// SIMATIC S7-200 SMART project (STEP 7-Micro/WIN SMART), CPU SR30

SYMBOL_TABLE 表格 1
真空值              VD200
温度值              VD204
罗茨启动真空设定         VD208
罗茨停机真空设定         VD212
温度报警设定           VD216
温度急停设定           VD220
目标真空             VD224
螺杆电流值            VD228
开启清洗电流设定         VD232
关闭清洗电流设定         VD236
频率读取             VW100
电流读取             VW102
频率显示             VW104
电流显示             VW106
频率写入             VW108
手动频率             VW110
清洗时间设定           VW112
吹扫时间设定           VW114
清洗时间显示           VW116
吹扫时间显示           VW118
清洗时间中间量          VW120
吹扫时间中间量          VW122
自动步骤             VW20
延时定时器            T50
流量开关定时器          T51
清洗定时器            T37
吹扫定时器            T38
故障急停             V300.0
故障报警             V300.1
流量开关fault        V300.2
液位开关fault        V300.3
变频器fault         V300.4
罗茨风机过载fault      V300.5
螺杆过载fault        V300.6
急停fault          V300.7
高温报警fault        V301.0
高温急停fault        V301.1
螺杆泵HMI           V500.0
罗茨泵HMI           V500.1
入口阀HMI           V500.2
清洗阀HMI           V500.3
吹扫阀HMI           V500.4
屏蔽蜂鸣器            V500.5
在线清洗HMI          V500.6
END_SYMBOL_TABLE

SYMBOL_TABLE 系统符号
Always_On        SM0.0    // 始终接通
First_Scan_On    SM0.1    // 仅在第一个扫描周期时接通
Clock_1s         SM0.5    // 针对 1 s 的周期时间，时钟脉冲接通 0.5 s，断开 0.5 s.
END_SYMBOL_TABLE

SYMBOL_TABLE 表格 3
主站完成位            M0.0
启动读写功            M0.1
一读完成位            M2.1
一写完成位            M2.2
二读完成位            M2.3
二写完成位            M2.4
主站错误代            MB1
延时触发             M30.0
通讯心跳             M11.2
END_SYMBOL_TABLE

ORGANIZATION_BLOCK MAIN:OB1
TITLE=程序注释
BEGIN
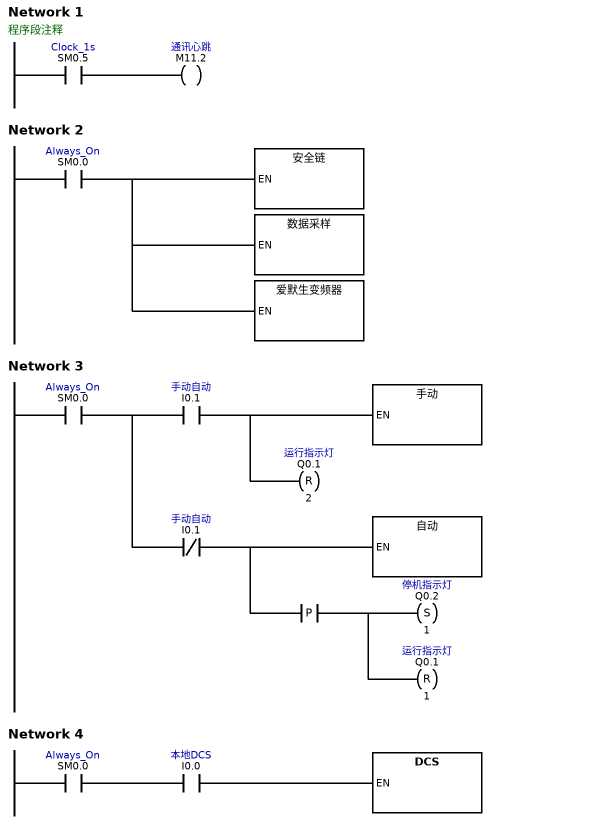
Network 1
// 程序段注释
LD     Clock_1s:SM0.5
=      通讯心跳:M11.2
Network 2
LD     Always_On:SM0.0
CALL   安全链:SBR2
CALL   数据采样:SBR1
CALL   爱默生变频器:SBR0
Network 3
LD     Always_On:SM0.0
LPS
A      手动自动:I0.1
CALL   手动:SBR3
R      运行指示灯:Q0.1, 2
LPP
AN     手动自动:I0.1
CALL   自动:SBR4
EU
S      停机指示灯:Q0.2, 1
R      运行指示灯:Q0.1, 1
Network 4
LD     Always_On:SM0.0
A      本地DCS:I0.0
CALL   DCS:SBR5
END_ORGANIZATION_BLOCK

SUBROUTINE_BLOCK 爱默生变频器:SBR0
TITLE=子程序注释
BEGIN
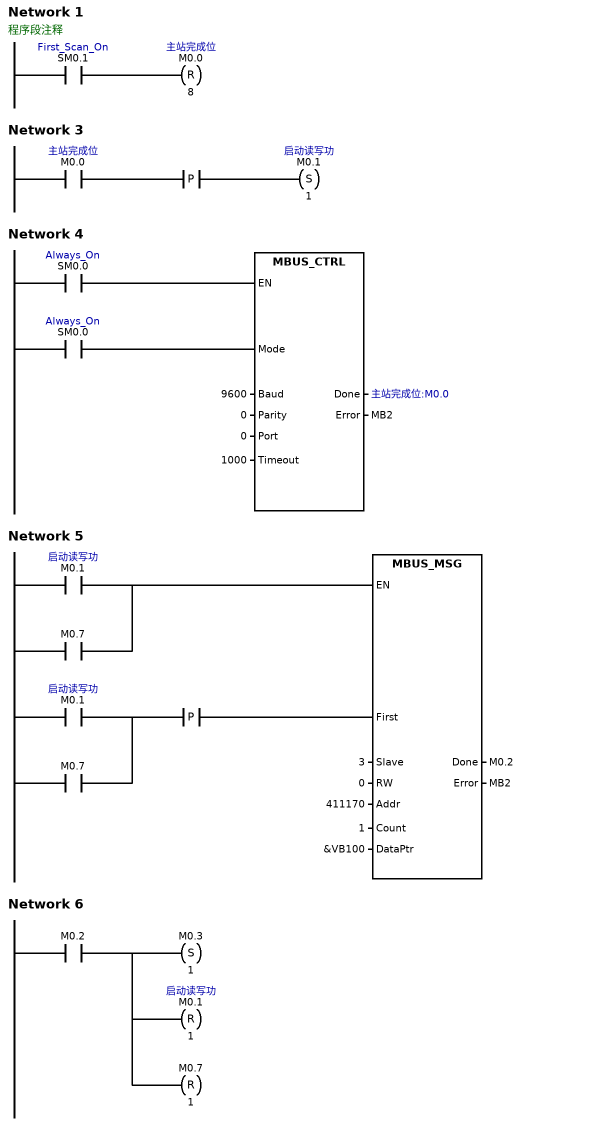
Network 1
// 程序段注释
LD     First_Scan_On:SM0.1
R      主站完成位:M0.0, 8
Network 3
LD     主站完成位:M0.0
EU
S      启动读写功:M0.1, 1
Network 4
LD     Always_On:SM0.0
=      L60.0
LD     Always_On:SM0.0
=      L63.7
LD     L60.0
CALL   MBUS_CTRL:SBR7, L63.7, 9600, 0, 0, 1000, 主站完成位:M0.0, MB2
Network 5
LD     启动读写功:M0.1
O      M0.7
=      L60.0
LD     启动读写功:M0.1
O      M0.7
EU
=      L63.7
LD     L60.0
CALL   MBUS_MSG:SBR8, L63.7, 3, 0, 411170, 1, &VB100, M0.2, MB2
Network 6
LD     M0.2
S      M0.3, 1
R      启动读写功:M0.1, 1
R      M0.7, 1
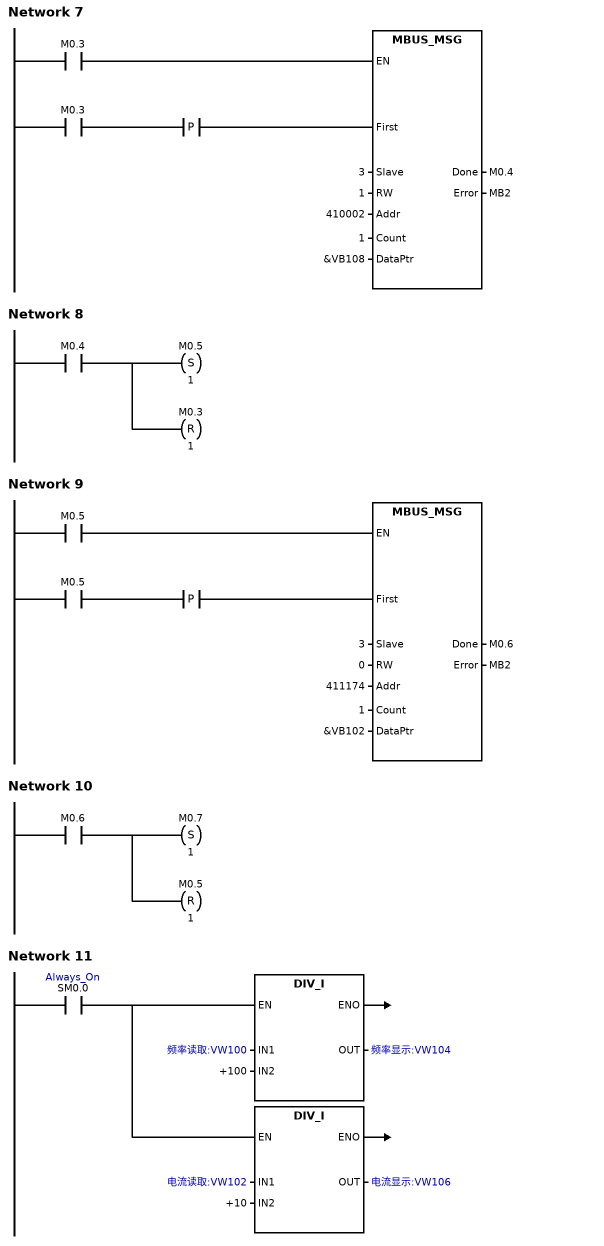
Network 7
LD     M0.3
=      L60.0
LD     M0.3
EU
=      L63.7
LD     L60.0
CALL   MBUS_MSG:SBR8, L63.7, 3, 1, 410002, 1, &VB108, M0.4, MB2
Network 8
LD     M0.4
S      M0.5, 1
R      M0.3, 1
Network 9
LD     M0.5
=      L60.0
LD     M0.5
EU
=      L63.7
LD     L60.0
CALL   MBUS_MSG:SBR8, L63.7, 3, 0, 411174, 1, &VB102, M0.6, MB2
Network 10
LD     M0.6
S      M0.7, 1
R      M0.5, 1
Network 11
LD     Always_On:SM0.0
MOVW   频率读取:VW100, 频率显示:VW104
/I     +100, 频率显示:VW104
MOVW   电流读取:VW102, 电流显示:VW106
/I     +10, 电流显示:VW106
END_SUBROUTINE_BLOCK

SUBROUTINE_BLOCK 数据采样:SBR1
TITLE=子程序注释
BEGIN
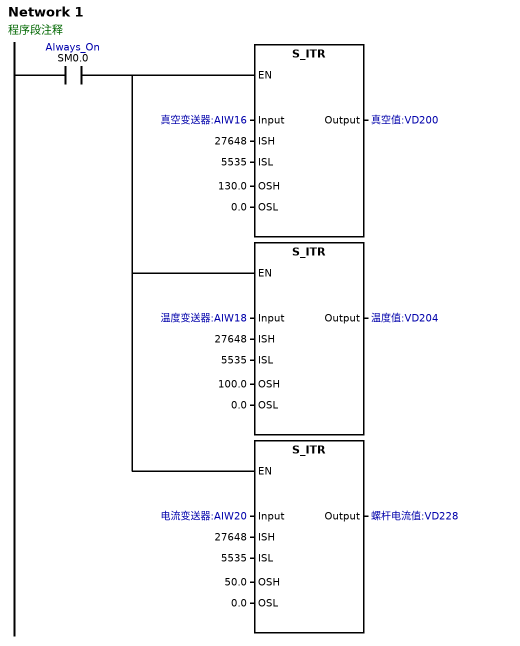
Network 1
// 程序段注释
LD     Always_On:SM0.0
CALL   S_ITR:SBR6, 真空变送器:AIW16, 27648, 5535, 130.0, 0.0, 真空值:VD200
CALL   S_ITR:SBR6, 温度变送器:AIW18, 27648, 5535, 100.0, 0.0, 温度值:VD204
CALL   S_ITR:SBR6, 电流变送器:AIW20, 27648, 5535, 50.0, 0.0, 螺杆电流值:VD228
END_SUBROUTINE_BLOCK

SUBROUTINE_BLOCK 安全链:SBR2
TITLE=子程序注释
BEGIN
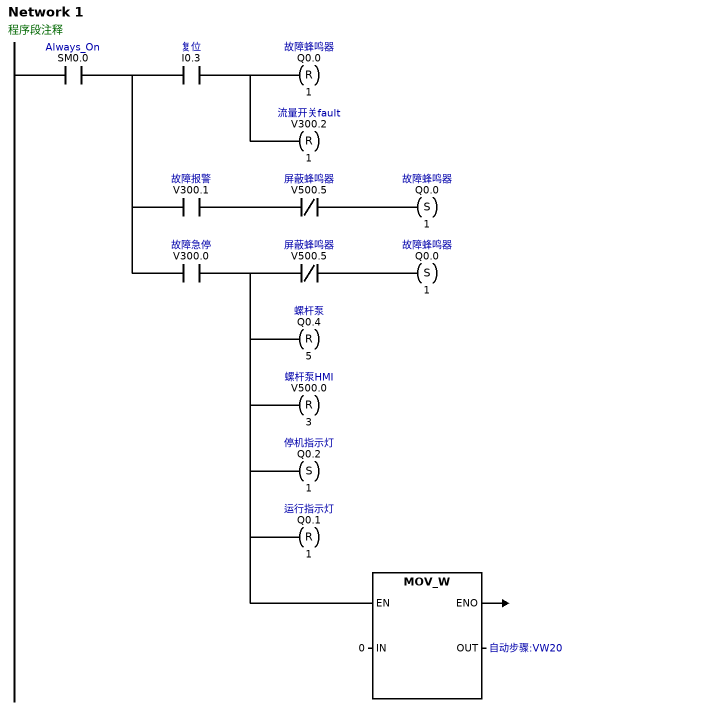
Network 1
// 程序段注释
LD     Always_On:SM0.0
LPS
A      复位:I0.3
R      故障蜂鸣器:Q0.0, 1
R      流量开关fault:V300.2, 1
LRD
A      故障报警:V300.1
AN     屏蔽蜂鸣器:V500.5
S      故障蜂鸣器:Q0.0, 1
LPP
A      故障急停:V300.0
LPS
AN     屏蔽蜂鸣器:V500.5
S      故障蜂鸣器:Q0.0, 1
LRD
R      螺杆泵:Q0.4, 5
LRD
R      螺杆泵HMI:V500.0, 3
LRD
S      停机指示灯:Q0.2, 1
LRD
R      运行指示灯:Q0.1, 1
LPP
MOVW   0, 自动步骤:VW20
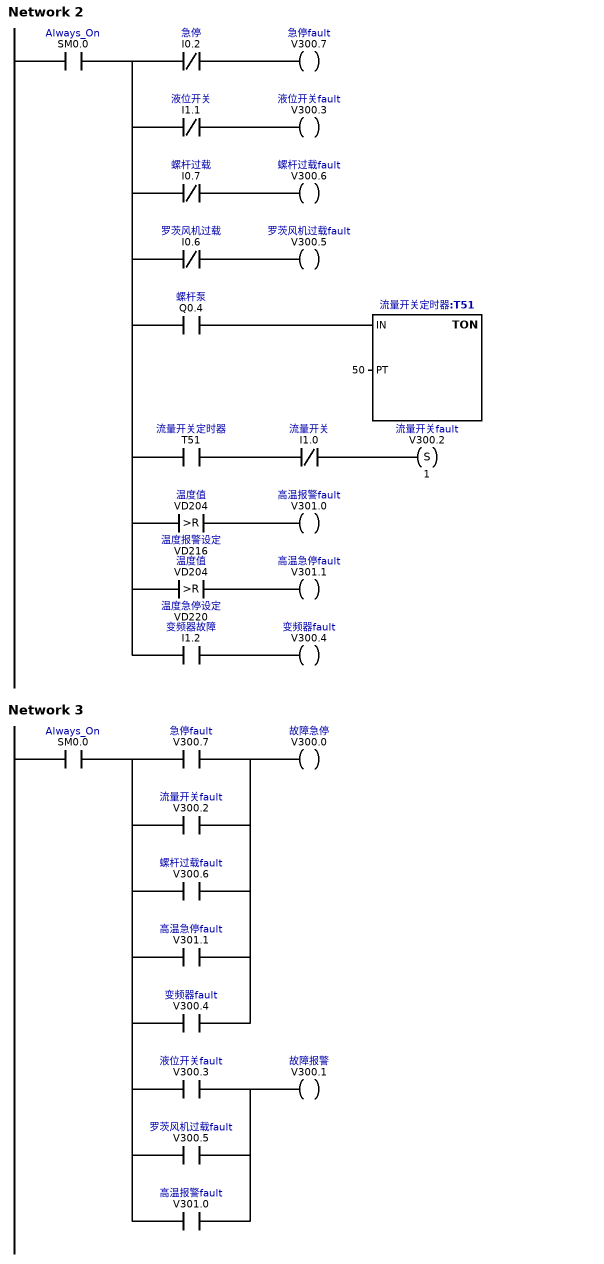
Network 2
LD     Always_On:SM0.0
LPS
AN     急停:I0.2
=      急停fault:V300.7
LRD
AN     液位开关:I1.1
=      液位开关fault:V300.3
LRD
AN     螺杆过载:I0.7
=      螺杆过载fault:V300.6
LRD
AN     罗茨风机过载:I0.6
=      罗茨风机过载fault:V300.5
LRD
A      螺杆泵:Q0.4
TON    流量开关定时器:T51, 50
LRD
A      流量开关定时器:T51
AN     流量开关:I1.0
S      流量开关fault:V300.2, 1
LRD
AR>    温度值:VD204, 温度报警设定:VD216
=      高温报警fault:V301.0
LRD
AR>    温度值:VD204, 温度急停设定:VD220
=      高温急停fault:V301.1
LPP
A      变频器故障:I1.2
=      变频器fault:V300.4
Network 3
LD     Always_On:SM0.0
LPS
LD     急停fault:V300.7
O      流量开关fault:V300.2
O      螺杆过载fault:V300.6
O      高温急停fault:V301.1
O      变频器fault:V300.4
ALD
=      故障急停:V300.0
LPP
LD     液位开关fault:V300.3
O      罗茨风机过载fault:V300.5
O      高温报警fault:V301.0
ALD
=      故障报警:V300.1
END_SUBROUTINE_BLOCK

SUBROUTINE_BLOCK 手动:SBR3
TITLE=子程序注释
BEGIN
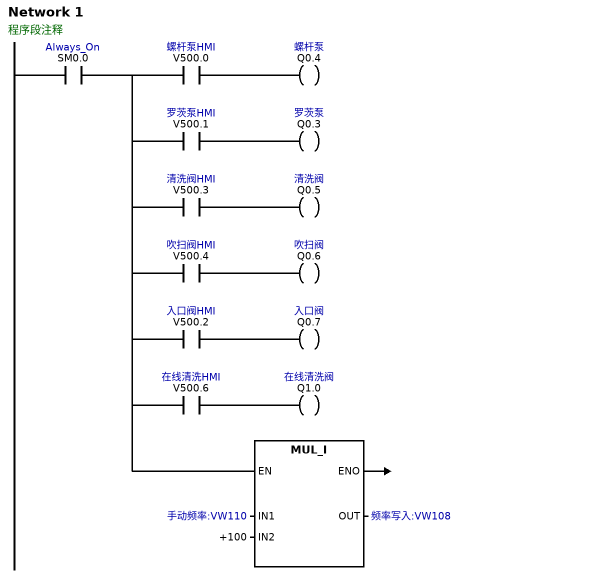
Network 1
// 程序段注释
LD     Always_On:SM0.0
LPS
A      螺杆泵HMI:V500.0
=      螺杆泵:Q0.4
LRD
A      罗茨泵HMI:V500.1
=      罗茨泵:Q0.3
LRD
A      清洗阀HMI:V500.3
=      清洗阀:Q0.5
LRD
A      吹扫阀HMI:V500.4
=      吹扫阀:Q0.6
LRD
A      入口阀HMI:V500.2
=      入口阀:Q0.7
LRD
A      在线清洗HMI:V500.6
=      在线清洗阀:Q1.0
LPP
MOVW   手动频率:VW110, 频率写入:VW108
*I     +100, 频率写入:VW108
END_SUBROUTINE_BLOCK

SUBROUTINE_BLOCK 自动:SBR4
TITLE=子程序注释
BEGIN
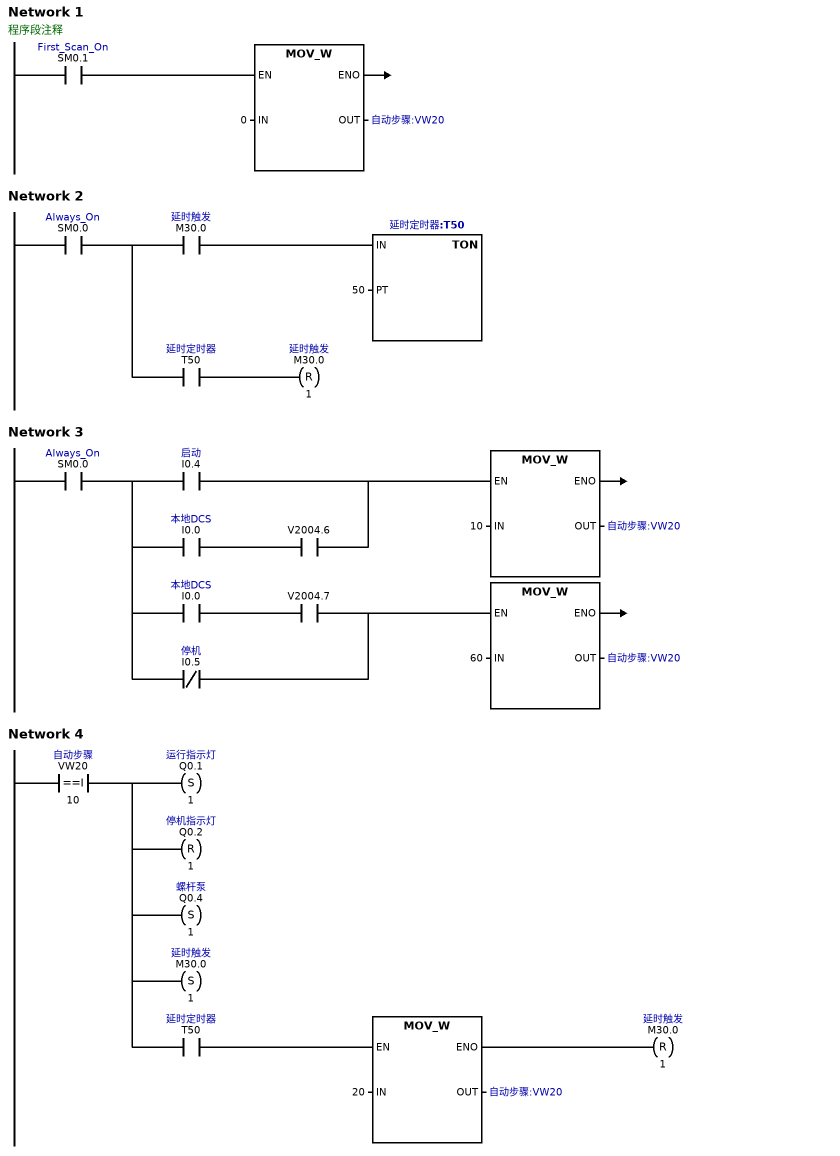
Network 1
// 程序段注释
LD     First_Scan_On:SM0.1
MOVW   0, 自动步骤:VW20
Network 2
LD     Always_On:SM0.0
LPS
A      延时触发:M30.0
TON    延时定时器:T50, 50
LPP
A      延时定时器:T50
R      延时触发:M30.0, 1
Network 3
LD     Always_On:SM0.0
LPS
LD     启动:I0.4
LD     本地DCS:I0.0
A      V2004.6
OLD
ALD
MOVW   10, 自动步骤:VW20
LPP
LD     本地DCS:I0.0
A      V2004.7
ON     停机:I0.5
ALD
MOVW   60, 自动步骤:VW20
Network 4
LDW=   自动步骤:VW20, 10
S      运行指示灯:Q0.1, 1
R      停机指示灯:Q0.2, 1
S      螺杆泵:Q0.4, 1
S      延时触发:M30.0, 1
A      延时定时器:T50
MOVW   20, 自动步骤:VW20
AENO
R      延时触发:M30.0, 1
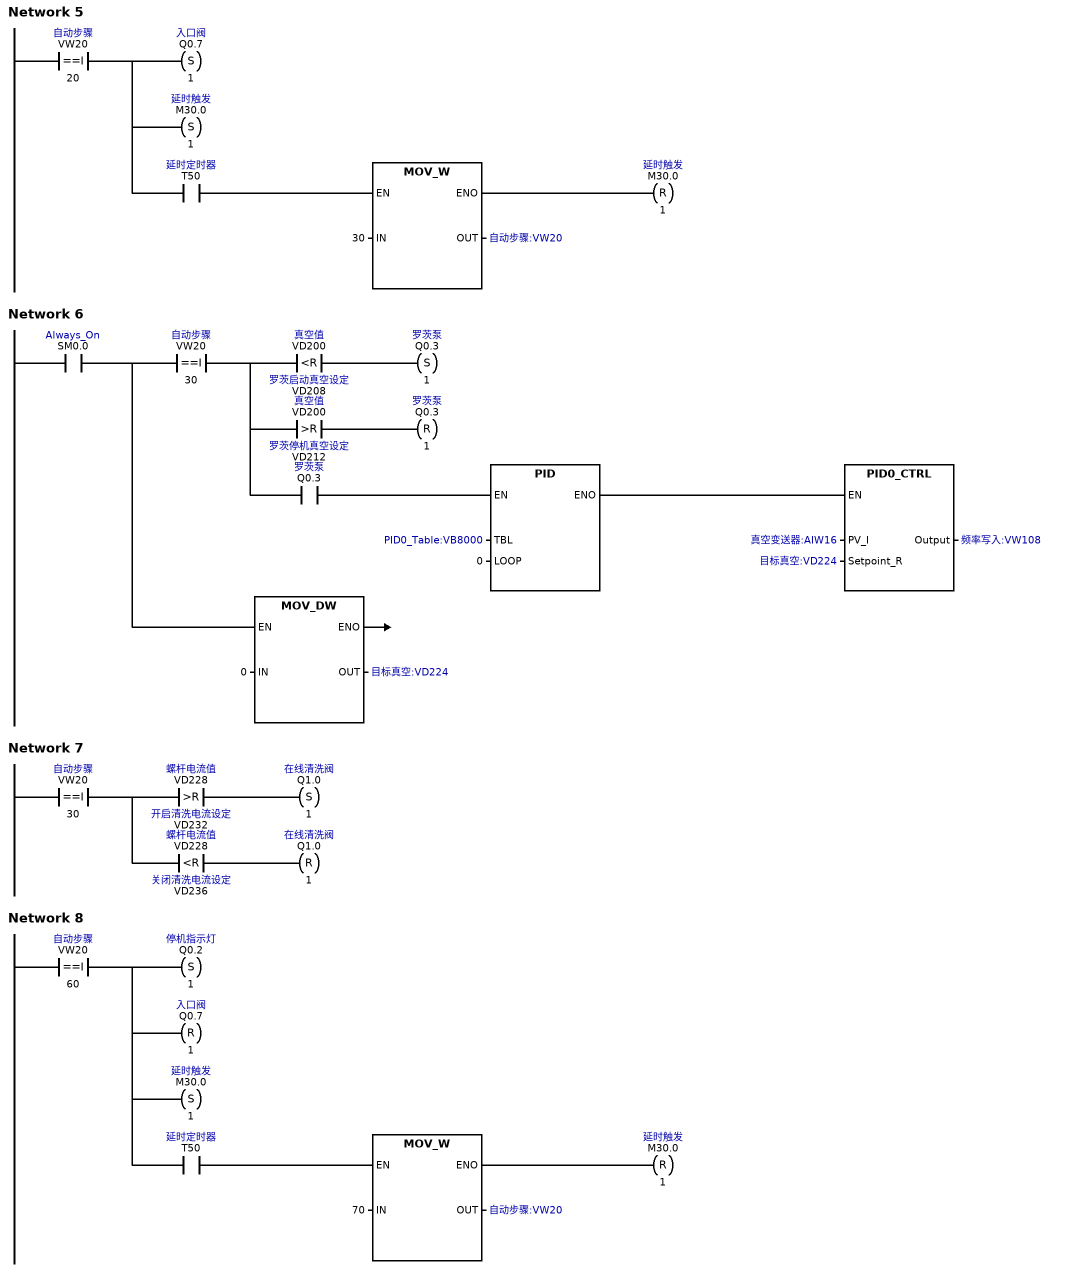
Network 5
LDW=   自动步骤:VW20, 20
S      入口阀:Q0.7, 1
S      延时触发:M30.0, 1
A      延时定时器:T50
MOVW   30, 自动步骤:VW20
AENO
R      延时触发:M30.0, 1
Network 6
LD     Always_On:SM0.0
LPS
AW=    自动步骤:VW20, 30
LPS
AR<    真空值:VD200, 罗茨启动真空设定:VD208
S      罗茨泵:Q0.3, 1
LRD
AR>    真空值:VD200, 罗茨停机真空设定:VD212
R      罗茨泵:Q0.3, 1
LPP
A      罗茨泵:Q0.3
PID    PID0_Table:VB8000, 0
AENO
CALL   PID0_CTRL:SBR10, 真空变送器:AIW16, 目标真空:VD224, 频率写入:VW108
LPP
MOVD   0, 目标真空:VD224
Network 7
LDW=   自动步骤:VW20, 30
LPS
AR>    螺杆电流值:VD228, 开启清洗电流设定:VD232
S      在线清洗阀:Q1.0, 1
LPP
AR<    螺杆电流值:VD228, 关闭清洗电流设定:VD236
R      在线清洗阀:Q1.0, 1
Network 8
LDW=   自动步骤:VW20, 60
S      停机指示灯:Q0.2, 1
R      入口阀:Q0.7, 1
S      延时触发:M30.0, 1
A      延时定时器:T50
MOVW   70, 自动步骤:VW20
AENO
R      延时触发:M30.0, 1
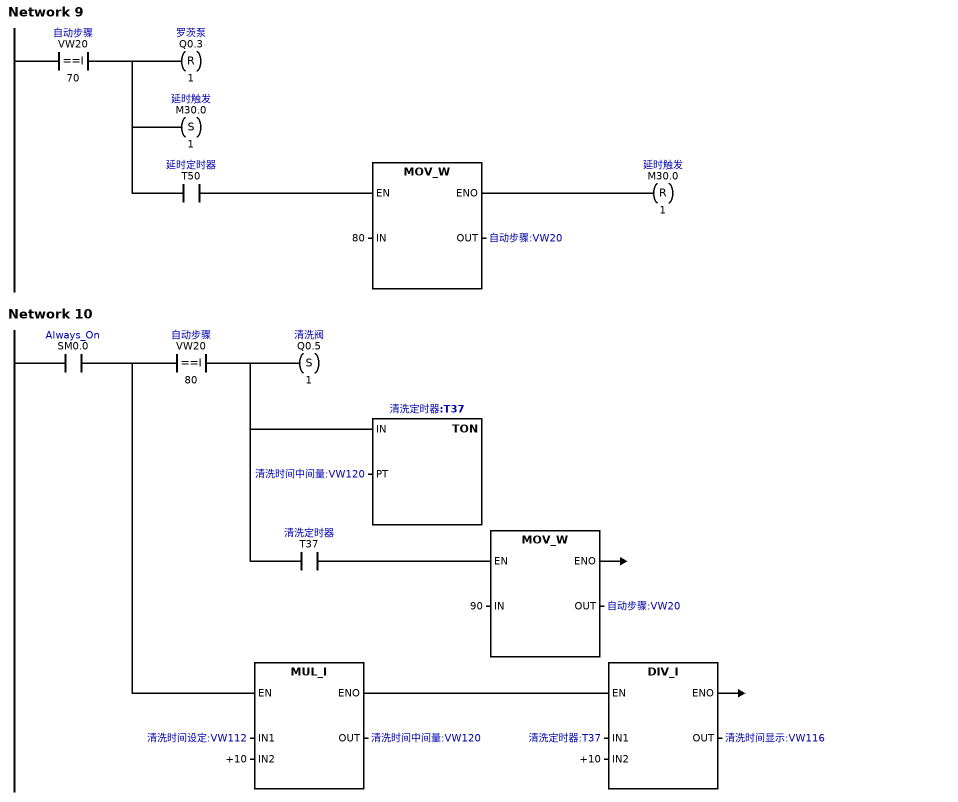
Network 9
LDW=   自动步骤:VW20, 70
R      罗茨泵:Q0.3, 1
S      延时触发:M30.0, 1
A      延时定时器:T50
MOVW   80, 自动步骤:VW20
AENO
R      延时触发:M30.0, 1
Network 10
LD     Always_On:SM0.0
LPS
AW=    自动步骤:VW20, 80
S      清洗阀:Q0.5, 1
TON    清洗定时器:T37, 清洗时间中间量:VW120
A      清洗定时器:T37
MOVW   90, 自动步骤:VW20
LPP
MOVW   清洗时间设定:VW112, 清洗时间中间量:VW120
AENO
*I     +10, 清洗时间中间量:VW120
AENO
MOVW   清洗定时器:T37, 清洗时间显示:VW116
/I     +10, 清洗时间显示:VW116
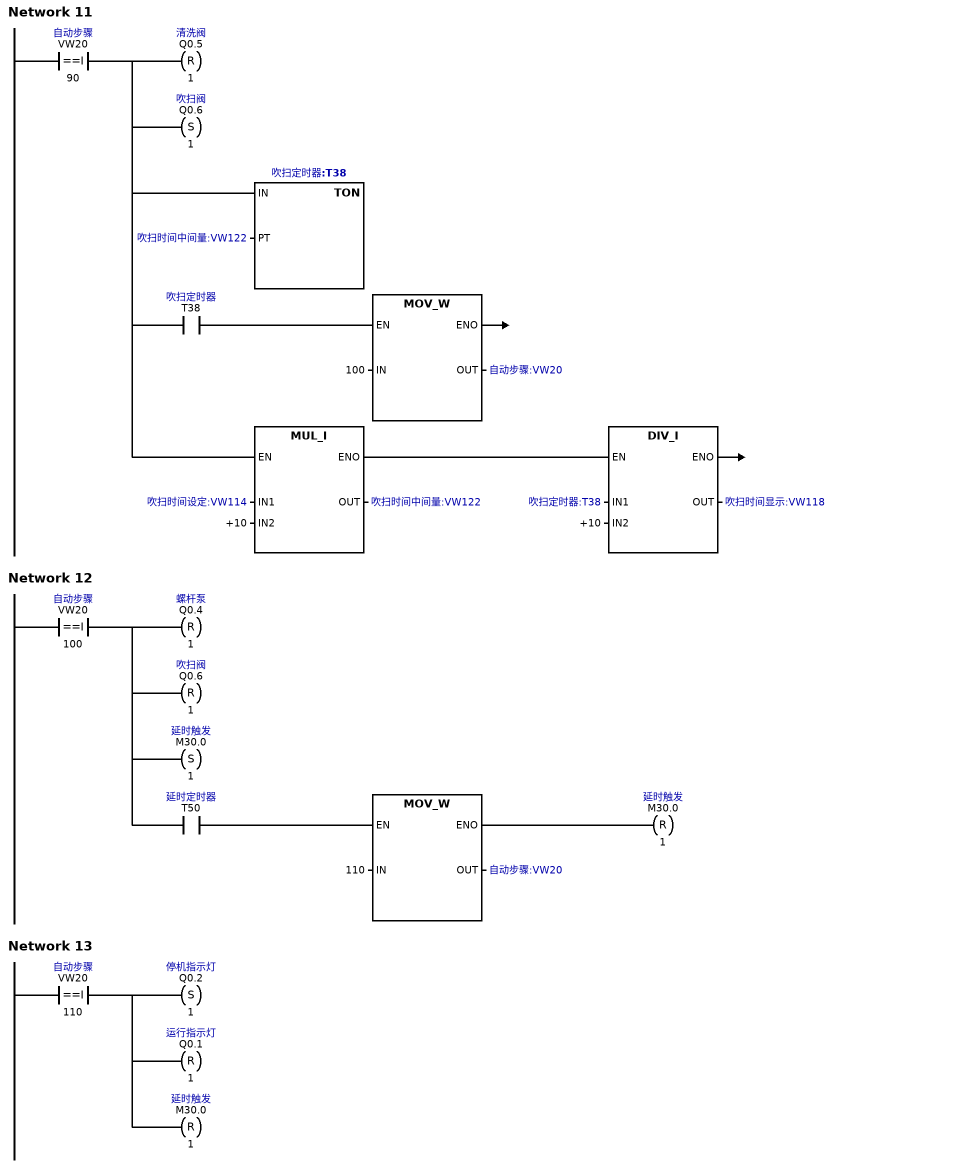
Network 11
LDW=   自动步骤:VW20, 90
LPS
R      清洗阀:Q0.5, 1
S      吹扫阀:Q0.6, 1
TON    吹扫定时器:T38, 吹扫时间中间量:VW122
A      吹扫定时器:T38
MOVW   100, 自动步骤:VW20
LPP
MOVW   吹扫时间设定:VW114, 吹扫时间中间量:VW122
AENO
*I     +10, 吹扫时间中间量:VW122
AENO
MOVW   吹扫定时器:T38, 吹扫时间显示:VW118
/I     +10, 吹扫时间显示:VW118
Network 12
LDW=   自动步骤:VW20, 100
R      螺杆泵:Q0.4, 1
R      吹扫阀:Q0.6, 1
S      延时触发:M30.0, 1
A      延时定时器:T50
MOVW   110, 自动步骤:VW20
AENO
R      延时触发:M30.0, 1
Network 13
LDW=   自动步骤:VW20, 110
S      停机指示灯:Q0.2, 1
R      运行指示灯:Q0.1, 1
R      延时触发:M30.0, 1
END_SUBROUTINE_BLOCK

SUBROUTINE_BLOCK DCS:SBR5
TITLE=子程序注释
BEGIN
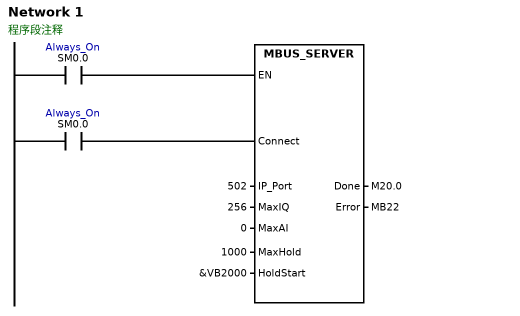
Network 1
// 程序段注释
LD     Always_On:SM0.0
=      L60.0
LD     Always_On:SM0.0
=      L63.7
LD     L60.0
CALL   MBUS_SERVER:SBR14, L63.7, 502, 256, 0, 1000, &VB2000, M20.0, MB22
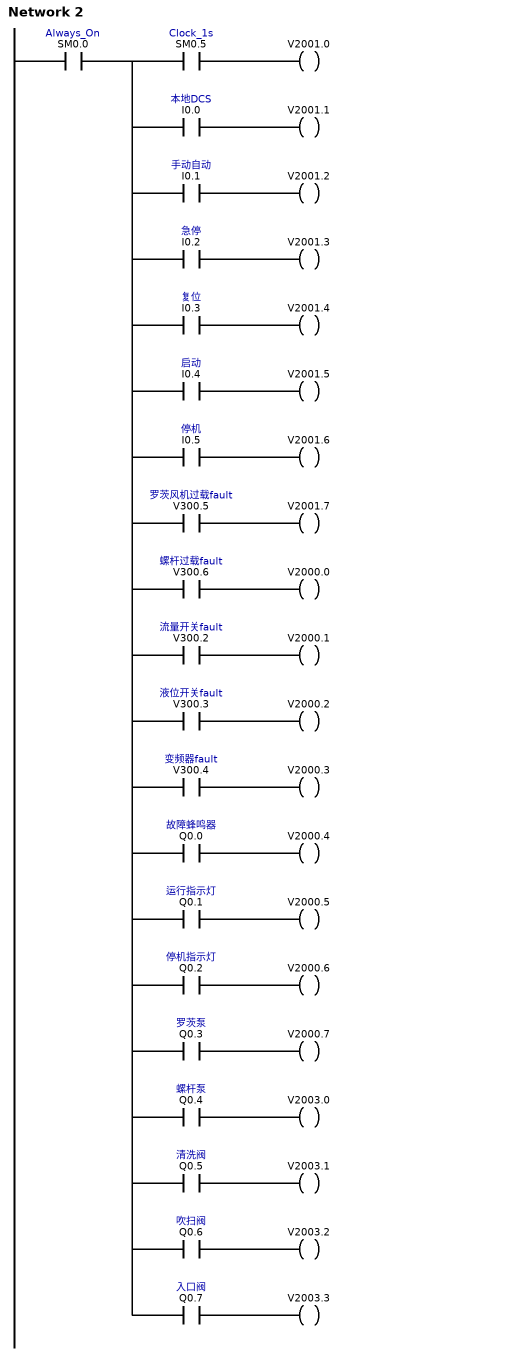
Network 2
LD     Always_On:SM0.0
LPS
A      Clock_1s:SM0.5
=      V2001.0
LRD
A      本地DCS:I0.0
=      V2001.1
LRD
A      手动自动:I0.1
=      V2001.2
LRD
A      急停:I0.2
=      V2001.3
LRD
A      复位:I0.3
=      V2001.4
LRD
A      启动:I0.4
=      V2001.5
LRD
A      停机:I0.5
=      V2001.6
LRD
A      罗茨风机过载fault:V300.5
=      V2001.7
LRD
A      螺杆过载fault:V300.6
=      V2000.0
LRD
A      流量开关fault:V300.2
=      V2000.1
LRD
A      液位开关fault:V300.3
=      V2000.2
LRD
A      变频器fault:V300.4
=      V2000.3
LRD
A      故障蜂鸣器:Q0.0
=      V2000.4
LRD
A      运行指示灯:Q0.1
=      V2000.5
LRD
A      停机指示灯:Q0.2
=      V2000.6
LRD
A      罗茨泵:Q0.3
=      V2000.7
LRD
A      螺杆泵:Q0.4
=      V2003.0
LRD
A      清洗阀:Q0.5
=      V2003.1
LRD
A      吹扫阀:Q0.6
=      V2003.2
LPP
A      入口阀:Q0.7
=      V2003.3
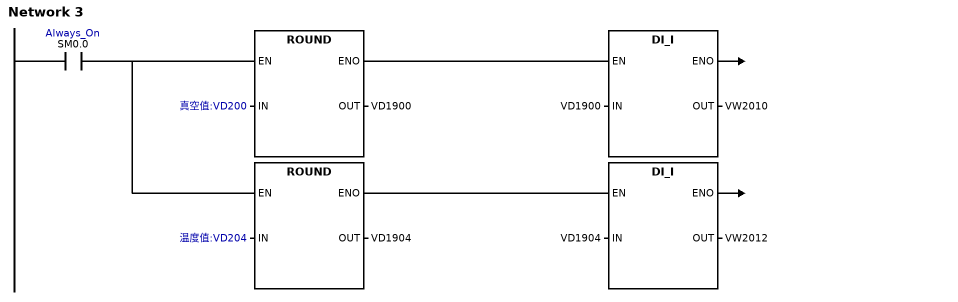
Network 3
LD     Always_On:SM0.0
LPS
ROUND  真空值:VD200, VD1900
AENO
DTI    VD1900, VW2010
LPP
ROUND  温度值:VD204, VD1904
AENO
DTI    VD1904, VW2012
END_SUBROUTINE_BLOCK

// SBR6: protected block, not included

// SBR7: protected block, not included

// SBR8: protected block, not included

// SBR9: protected block, not included

// SBR10: protected block, not included

// SBR11: protected block, not included

// SBR12: protected block, not included

// SBR13: protected block, not included

// SBR14: protected block, not included
